// List collection implemeneted using a dynamic array.
{attribute 'enable_dynamic_creation'}
{attribute 'no_assign'}
{attribute 'no_explicit_call' := 'direct call for this function block is not allowed'}
FUNCTION_BLOCK FINAL FB_Array_List EXTENDS FB_Collection IMPLEMENTS I_Array_List//, I_Enumerable, I_Copyable
VAR
	pBuffer : POINTER TO T_Generic;
	Capacity : T_Capacity;
END_VAR

// Size of the storage space currently allocated for the array list.
PROPERTY FINAL _Capacity : T_Capacity
GET
_Capacity := THIS^.Capacity;
END_GET
SET // PROTECTED
THIS^.Capacity := _Capacity;
END_SET
END_PROPERTY

// Adds an item to the end of the list.
METHOD Append : I_List
VAR_INPUT
	Item : ANY; // Value to store in list
END_VAR
VAR_OUTPUT
	bSuccess : BOOL;
END_VAR
Append := THIS^;

THIS^.Insert_Generic(THIS^._Count, Item, bSuccess => bSuccess);
END_METHOD

// Empties/Clears/Deletes every item in the list.
METHOD Clear : I_List
VAR
	i : T_Capacity;
END_VAR
Clear := THIS^;

THIS^.Clear_Error();

IF THIS^._Is_Empty THEN RETURN; END_IF
IF THIS^.pBuffer = 0 THEN RETURN; END_IF

FOR i := 0 TO THIS^._Count - 1 DO
	F_Delete_Generic(THIS^.pBuffer[i]);
	END_FOR
	
THIS^._Count := 0;
END_METHOD

// Checks if item is contained in list.
METHOD Contains : BOOL
VAR_INPUT
	Item : ANY; // Item to find in list
END_VAR
THIS^.Search(Item, bSuccess => Contains);
END_METHOD

{attribute 'hide'}
METHOD FB_exit : BOOL
VAR_INPUT
	bInCopyCode : BOOL; // if TRUE, the exit method is called for exiting an instance that is copied afterwards (online change).
END_VAR
// Return if it's an online change.
IF bInCopyCode OR_ELSE THIS^.pBuffer = 0 THEN RETURN; END_IF

THIS^.Clear();
__DELETE(THIS^.pBuffer);
THIS^._Capacity := 0;
END_METHOD

{attribute 'hide'}
METHOD FB_init : BOOL
VAR_INPUT
	bInitRetains 		: BOOL; // if TRUE, the retain variables are initialized (warm start / cold start)
	bInCopyCode 		: BOOL; // if TRUE, the instance afterwards gets moved into the copy code (online change)
	Initial_Capacity 	: T_Capacity; // The capacity and count to initialise the array list with.
END_VAR
VAR 
	i : T_Capacity;
END_VAR
// Return if it's an online change.
IF bInCopyCode THEN RETURN; END_IF

THIS^.FB_exit(0);
THIS^.Resize(Initial_Capacity);
THIS^._Count := Initial_Capacity;


IF THIS^._Is_Empty THEN RETURN; END_IF

FOR i := 0 TO THIS^._Count - 1 DO
	THIS^.pBuffer[i].TypeClass := T_Type.TYPE_NONE;
	END_FOR
END_METHOD

// Gets item from list at specified location without removing it
METHOD Get : I_List
VAR_INPUT
	Index : T_Position; // Location of item
	Item : ANY;  // Variable to store returned item
END_VAR
VAR_OUTPUT
	bSuccess : BOOL;
END_VAR
Get := THIS^;

IF Index < 0 OR_ELSE Index >= THIS^._Count THEN
	THIS^._Error_Status := F_Error(TRUE, GVL_Errors.ERR_OUT_OF_LIMITS, 'Index out of bounds.');
	RETURN;
	END_IF

IF NOT F_Matching_Generics(Item, THIS^.pBuffer[Index]) THEN
	THIS^._Error_Status := F_Error(TRUE, GVL_Errors.ERR_TYPE_MISMATCH, 'Type mismatch.');
	RETURN;
	END_IF
	
F_Copy_Generic_Value(THIS^.pBuffer[Index], Item);
bSuccess := TRUE;
THIS^.Clear_Error();
END_METHOD

// Returns item as a string, if type to string conversion is supported
METHOD Get_As_String : I_List
VAR_INPUT
	Index : T_Position; // Location of item
	sItem : REFERENCE TO STRING; // Variable to store returned item.
END_VAR
VAR_OUTPUT
	bSuccess : BOOL;
END_VAR
Get_As_String := THIS^;

IF NOT __ISVALIDREF(sItem) THEN 
	THIS^._Error_Status := F_Error(TRUE, GVL_Errors.ERR_INVALID_REFERENCE, 'Invalid reference.');
	RETURN;
	END_IF

IF Index < 0 OR_ELSE Index >= THIS^._Count THEN
	THIS^._Error_Status := F_Error(TRUE, GVL_Errors.ERR_OUT_OF_LIMITS, 'Index out of bounds.');
	RETURN;
	END_IF
	
IF NOT F_String_Convertable_Generic(THIS^.pBuffer[Index]) THEN 
	THIS^._Error_Status := F_Error(TRUE, GVL_Errors.ERR_NOT_SUPPORTED, 'No support for converting item at index to string.');
	RETURN;
	END_IF
	
CASE THIS^.pBuffer[Index].TypeClass OF
	T_Type.TYPE_STRING:
		Tc2_Utilities.STRNCPY(ADR(sItem), THIS^.pBuffer[Index].pValue, MIN(Tc2_Utilities.LEN2(ADR(sItem))+1, TO_UDINT(THIS^.pBuffer[Index].diSize)));

	T_Type.TYPE_WSTRING:
		Tc2_Utilities.WSTRING_TO_STRING2(ADR(sItem), THIS^.pBuffer[Index].pValue, MIN(Tc2_Utilities.LEN2(ADR(sItem))+1, TO_UDINT(THIS^.pBuffer[Index].diSize)));
ELSE
	sItem := F_Generic_To_String(THIS^.pBuffer[Index]);
	END_CASE
	
bSuccess := TRUE;
THIS^.Clear_Error();
END_METHOD

// Gets a value from a list in it's generic form.
// (** Use carefully as this contains the pointer of the actual value in the collection. **)
// If you wish to use this it is recommeded you create a copy of the returned value using MEMMOVE or MEMCPY
METHOD Get_Generic : I_List
VAR_INPUT
	Index : T_Position; // Location of item
END_VAR
VAR_OUTPUT
	Item : T_Generic := (TypeClass := T_Type.TYPE_NONE);
	bSuccess : BOOL;
END_VAR
Get_Generic := THIS^;

IF Index < 0 OR_ELSE Index >= THIS^._Count THEN
	THIS^._Error_Status := F_Error(TRUE, GVL_Errors.ERR_OUT_OF_LIMITS, 'Index out of bounds.');
	RETURN;
	END_IF

Item := THIS^.pBuffer[Index];
bSuccess := TRUE;
THIS^.Clear_Error();
END_METHOD

// Gets the type of the item at specified location.
METHOD Get_Type_At : I_List
VAR_INPUT
	Index : T_Position;
END_VAR
VAR_OUTPUT
	Item_Type : T_Type := T_Type.TYPE_NONE;
	bSuccess : BOOL;
END_VAR
VAR
	Tmp : T_Generic;
END_VAR
Get_Type_At := THIS^;

THIS^.Get_Generic(Index, Item => Tmp, bSuccess => bSuccess);

IF bSuccess THEN Item_Type := Tmp.TypeClass; END_IF
END_METHOD

// Adds new item to list at specified location, if index = 0, item will be added at the front, if index = count, item will be added at the back
METHOD Insert : I_List
VAR_INPUT
	Index : T_Position; // Location of item
	Item : ANY; // Item to store in list
END_VAR
VAR_OUTPUT
	bSuccess : BOOL;
END_VAR
Insert := THIS^;
THIS^.Insert_Generic(Index, Item, bSuccess => bSuccess);
END_METHOD

// Adds new item to list at specified location using the generic form. 
// If index = 0, item will be added at the front, if index = count, item will be added at the back
METHOD Insert_Generic : I_List
VAR_INPUT
	Index 	 : T_Position; 	// Location of item
	Item 	 : T_Generic;  	// Item to store in list
END_VAR
VAR_OUTPUT
	bSuccess : BOOL;
END_VAR
Insert_Generic := THIS^;

IF THIS^._Count >= THIS^._Capacity THEN THIS^.Resize((THIS^._Count * 2) + 1); END_IF

IF Index = THIS^._Count THEN 
	// Add to back
	THIS^.pBuffer[THIS^._Count] := F_Clone_Generic(Item);
	THIS^.Increment_Count();
	bSuccess := TRUE;
	THIS^.Clear_Error();
	RETURN;
	END_IF

IF Index < 0 OR_ELSE Index > THIS^._Count THEN
	// Throw out of bounds error.
	THIS^._Error_Status := F_Error(TRUE, GVL_Errors.ERR_OUT_OF_LIMITS, 'Index out of bounds.');
	RETURN;
	END_IF
	
Tc2_System.MEMMOVE(ADR(THIS^.pBuffer[Index + 1]), ADR(THIS^.pBuffer[Index]), TO_UDINT((THIS^._Count - Index) * SIZEOF(T_Generic)));
THIS^.pBuffer[Index] := F_Clone_Generic(Item);
THIS^.Increment_Count();
bSuccess := TRUE;
THIS^.Clear_Error();
END_METHOD

// Adds an item at the front of the list.
METHOD Prepend : I_List
VAR_INPUT
	Item : ANY; // Value to store in list
END_VAR
VAR_OUTPUT
	bSuccess : BOOL;
END_VAR
Prepend := THIS^;

THIS^.Insert_Generic(0, Item, bSuccess => bSuccess);
END_METHOD

// Removes item from the list.
METHOD Remove : I_List
VAR_INPUT
	Item : ANY; // Item to remove from in list
END_VAR
VAR_OUTPUT
	bSuccess : BOOL;
END_VAR
VAR
	Tmp : T_Position;
END_VAR
Remove := THIS^;

THIS^.Search(Item, Index => Tmp, bSuccess => bSuccess);
IF NOT bSuccess THEN RETURN; END_IF 
THIS^.Remove_At(0, bSuccess => bSuccess);
END_METHOD

// Remove item at specified location 
METHOD Remove_At : I_List
VAR_INPUT
	Index : T_Position; // Location of item
END_VAR
VAR_OUTPUT
	bSuccess : BOOL;
END_VAR
Remove_At := THIS^;

IF Index < 0 OR_ELSE Index >= THIS^._Count THEN
	THIS^._Error_Status := F_Error(TRUE, GVL_Errors.ERR_OUT_OF_LIMITS, 'Index out of bounds.');
	RETURN;
	END_IF


F_Delete_Generic(THIS^.pBuffer[Index]);	
Tc2_System.MEMMOVE(ADR(THIS^.pBuffer[Index]), ADR(THIS^.pBuffer[Index+1]), TO_UDINT(SIZEOF(T_Generic)*(THIS^._Count - Index - 1)));
THIS^.Decrement_Count();

IF THIS^._Count <= (THIS^._Capacity/4) THEN THIS^.Resize(THIS^._Capacity/2); END_IF

bSuccess := TRUE;
THIS^.Clear_Error();
END_METHOD

// Removes item at the back of the list.
METHOD Remove_Last : I_List
VAR_OUTPUT
	bSuccess : BOOL;
END_VAR
Remove_Last := THIS^.Remove_At(THIS^._Count - 1, bSuccess => bSuccess);
END_METHOD

// Manually resize list. If list becomes smaller, item on higher locations will be deleted.
METHOD Resize : I_List
VAR_INPUT
	Size : T_Capacity; // New size of list.
END_VAR
VAR_OUTPUT
	bSuccess : BOOL;
END_VAR
VAR
	pNew_Buffer : POINTER TO T_Generic;
	i, Number_Of_Elements_To_Copy : T_Capacity;
END_VAR
Resize := THIS^;

IF Size = 0 THEN THIS^.FB_exit(FALSE); bSuccess := TRUE; RETURN; END_IF
IF THIS^.pBuffer = 0 THEN THIS^.pBuffer := F_Malloc_Generic(1); THIS^._Capacity := 1; END_IF

pNew_Buffer := F_Malloc_Generic(Size);

Tc2_System.MEMCPY(pNew_Buffer, THIS^.pBuffer, TO_UDINT(SIZEOF(T_Generic)*THIS^._Count));

IF Size < THIS^._Count THEN
	FOR i := Size TO THIS^._Count - 1 DO F_Delete_Generic(THIS^.pBuffer[i]); END_FOR
	THIS^._Count := Size;
	END_IF

THIS^._Capacity := Size;

__DELETE(THIS^.pBuffer);
THIS^.pBuffer := pNew_Buffer;

bSuccess := TRUE;
THIS^.Clear_Error();
END_METHOD

// Reverses the order of items in the list
METHOD Reverse : I_List
VAR_OUTPUT
	bSuccess : BOOL;
END_VAR
VAR
	i : T_Capacity;
END_VAR
Reverse := THIS^;

IF NOT THIS^._Is_Empty THEN
	FOR i := 0 TO (THIS^._Count/2) - 1 DO
		F_Swap_Generics(THIS^.pBuffer[i], THIS^.pBuffer[THIS^._Count - i - 1]);
		END_FOR
	END_IF

bSuccess := TRUE;
THIS^.Clear_Error();
END_METHOD

// Find the location of an item in list.
METHOD Search : I_List
VAR_INPUT
	Item : ANY; // Item to find in list
END_VAR
VAR_OUTPUT
	Index : T_Position := -1; //Location of item in list 
	bSuccess : BOOL;
END_VAR
VAR
	i : T_Position;
END_VAR
Search := THIS^;

IF THIS^._Is_Empty THEN RETURN; END_IF
FOR i := 0 TO THIS^._Count - 1 DO
	CASE F_Compare_Generics(Item, THIS^.pBuffer[i]) OF
		T_Comparison.Equal:
			bSuccess := TRUE;
			THIS^.Clear_Error();
			Index := i;
			RETURN;
		END_CASE
	END_FOR
	
THIS^._Error_Status := F_Error(TRUE, GVL_Errors.ERR_NO_OBJECT, 'Item not found.');
END_METHOD

// Changes the item at the specified location in the list.
METHOD Set : I_List
VAR_INPUT
	Index 	: T_Position; // Location of item
	Item 	: ANY; 	// Item to store in list
END_VAR
VAR_OUTPUT
	bSuccess : BOOL;
END_VAR
Set := THIS^;

THIS^.Set_Generic(Index, Item, bSuccess => bSuccess);
END_METHOD

// Changes the item at the specified location in the list in it's generic form.
METHOD Set_Generic : I_List
VAR_INPUT
	Index : T_Position; // Location of item
	Item : T_Generic;
END_VAR
VAR_OUTPUT
	bSuccess : BOOL;
END_VAR
Set_Generic := THIS^;

IF Index < 0 OR_ELSE Index >= THIS^._Count THEN
	THIS^._Error_Status := F_Error(TRUE, GVL_Errors.ERR_OUT_OF_LIMITS, 'Index out of bounds.');
	RETURN;
	END_IF
	
F_Delete_Generic(THIS^.pBuffer[Index]);
THIS^.pBuffer[Index] := F_Clone_Generic(Item);

bSuccess := TRUE;
THIS^.Clear_Error();
END_METHOD

// Swaps item at index A with item at index B.
METHOD Swap : I_List
VAR_INPUT
	Index_A, Index_B : T_Position;
END_VAR
VAR_OUTPUT
	bSuccess : BOOL;
END_VAR
Swap := THIS^;

IF Index_A < 0 OR_ELSE Index_A >= THIS^._Count OR_ELSE Index_B < 0 OR_ELSE Index_B >= THIS^._Count THEN
	THIS^._Error_Status := F_Error(TRUE, GVL_Errors.ERR_OUT_OF_LIMITS, 'Index out of bounds.');
	RETURN;
	END_IF
	
bSuccess := F_Swap_Generics(THIS^.pBuffer[Index_A], THIS^.pBuffer[Index_B]);
THIS^.Clear_Error();
END_METHOD

END_FUNCTION_BLOCK

(* stored: Version 1.1.0.1, ProductVersion 3.1.4024.4
   POU FB_Array_List: Id {1d0f1928-8b35-4b3e-b890-4196d49d0ef1}, SpecialFunc None
   Property _Capacity: Id {b081f4ac-2b87-4570-9185-414a607fec63}
   Get Get: Id {2a0bc92e-da23-4ff9-a372-f5fb4352723d}
   Set Set: Id {615296be-ab6d-4c7f-89e6-7db7c195512a}
   Method Append: Id {c0b24605-11f6-479b-a983-a79cd50031c8}
   Method Clear: Id {dbabc413-80fb-4b16-a01f-1bfc77e7d267}
   Method Contains: Id {90a090df-149d-4751-bd9b-d026d807973d}
   Method FB_exit: Id {f9bfb80b-da84-48a5-b521-af8424ca4753}
   Method FB_init: Id {da7d3329-ad02-4fd7-8e0d-4aaa794f99d7}
   Method Get: Id {39ea728c-38e0-44b4-88ce-acb9b7ab7dac}
   Method Get_As_String: Id {c7489442-0be9-490f-a0d5-753e7d2f05d2}
   Method Get_Generic: Id {a0fdc21c-e986-4996-b92d-e1185faedb99}
   Method Get_Type_At: Id {057ec36f-cff4-48a9-9e9a-3fff89515809}
   Method Insert: Id {87f490a7-b3c0-4c58-9c33-e5755fab7cbd}
   Method Insert_Generic: Id {13a183a2-9050-4198-9d56-f267da8a30f9}
   Method Prepend: Id {ac2a9b50-0f99-4d8d-824c-f56cc5087646}
   Method Remove: Id {a3aaf330-a3e6-4731-80e7-17c1a3f4154a}
   Method Remove_At: Id {f4e42044-e004-4f20-b51a-08fd45b15aff}
   Method Remove_Last: Id {59aaefa4-a54b-425a-9919-3bec50ac3826}
   Method Resize: Id {76fa8eb0-2d38-4b8a-b64f-9a86a8d9ddf4}
   Method Reverse: Id {7ac1c105-6985-4148-827d-da85bb707466}
   Method Search: Id {4dc2db7a-eeee-4cf0-9b03-32f7f83be003}
   Method Set: Id {2874a92a-c848-43b1-9a2b-b5425a9fd064}
   Method Set_Generic: Id {396d4717-01ca-4595-9a03-4199cd80b242}
   Method Swap: Id {094f7f81-8b07-4371-981d-f2985cfbd4e8} *)
